KUKA KRL program: wkz1_ab.src, wkz1_ab.dat

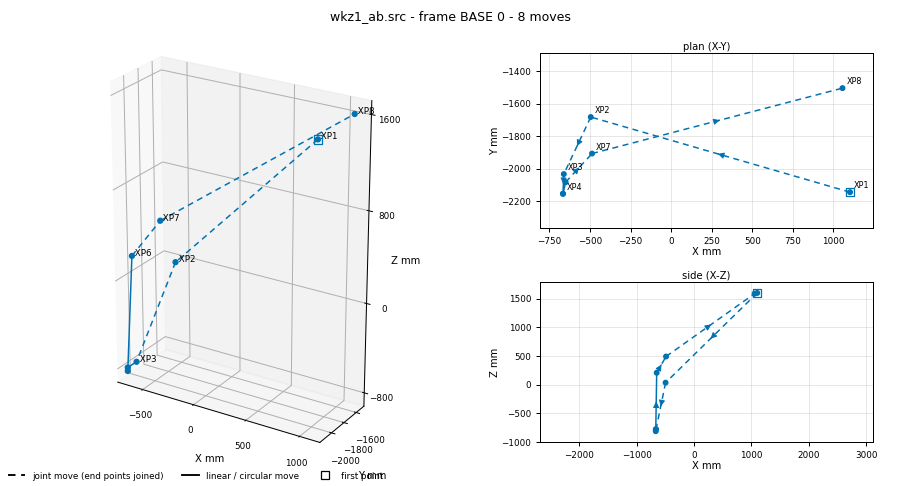
[picture p0: tool path of wkz1_ab.src in frame BASE 0, 8 of 8 moves have a stored position in this frame; points joined in program order, loops and branches not executed]
--- wkz1_ab.src ---
&ACCESS RVO8
&REL 103
&COMMENT DEP_C1
&PARAM DISKPATH = Program/WKZ
DEF WKZ1_AB ( )

;FOLD INI;%{PE}
  ;FOLD BASISTECH INI
    GLOBAL INTERRUPT DECL 3 WHEN $STOPMESS==TRUE DO IR_STOPM ( )
    INTERRUPT ON 3
    BAS (#INITMOV,0 )
  ;ENDFOLD (BASISTECH INI)
;FOLD SPOTTECH INI
USERSPOT(#INIT)
;ENDFOLD (SPOTTECH INI)
;FOLD GRIPPERTECH INI
USER_GRP(0,DUMMY,DUMMY,GDEFAULT)
;ENDFOLD (GRIPPERTECH INI)
  ;FOLD USER INI
    ;Make your modifications here

  ;ENDFOLD (USER INI)
;ENDFOLD (INI)
; Caracterização dos meios de produção:
; Versão Atual:
; 04/05/2013 12:00 Name: P13.090-R6 CHANGES: Deposita C1

chk_w1_wechs_ok ( )              ; CHECK GUN C1

;FOLD PTP P1 Vel=100 % PDAT1 Tool[1]:Gun C1 Base[0];%{PE}%R 8.2.24,%MKUKATPBASIS,%CMOVE,%VPTP,%P 1:PTP, 2:P1, 3:, 5:100, 7:PDAT1
$BWDSTART=FALSE
PDAT_ACT=PPDAT1
FDAT_ACT=FP1
BAS(#PTP_PARAMS,100)
PTP XP1
;ENDFOLD

;FOLD ; START INTERLOCK COM R4;%{PE}%R 8.2.24,%MKUKATPBASIS,%CCOMMENT,%VNORMAL,%P 2:START  INTERLOCK  COM  R4
;ENDFOLD
;FOLD Collision.Monitoring_4_On ;%{PE}%MKUKATPUSER

COLLSTOP( 4, 1 ) ;Interrupt-Controlled

;ENDFOLD

;FOLD WAIT FOR ( NOT IN 161 'DEPOSITO 1 OCUPADO' );%{PE}%R 8.2.24,%MKUKATPBASIS,%CEXT_WAIT_FOR,%VEXT_WAIT_FOR,%P 2:, 4:NOT, 5:$IN, 6:161, 7:DEPOSITO 1 OCUPADO, 9:
WAIT FOR  (  NOT $IN[161] )
;ENDFOLD
;FOLD WAIT FOR ( IN 219 'PLACA DE SUPORTE FUNDIDA' );%{PE}%R 8.2.24,%MKUKATPBASIS,%CEXT_WAIT_FOR,%VEXT_WAIT_FOR,%P 2:, 4:, 5:$IN, 6:219, 7:PLACA DE SUPORTE FUNDIDA, 9:
WAIT FOR  ( $IN[219] )
;ENDFOLD
;FOLD PULSE 167 'Proteção da pinca 1 abrir' State=TRUE Time=0.3 sec;%{PE}%R 8.2.24,%MKUKATPBASIS,%COUT,%VPULSE,%P 2:167, 3:Proteção da pinca 1 abrir, 5:TRUE, 6:, 8:0.3
PULSE($OUT[167], TRUE,0.3)
;ENDFOLD
;FOLD PULSE 184 'Proteção da pinca 3 fechar' State=TRUE Time=0.3 sec;%{PE}%R 8.2.24,%MKUKATPBASIS,%COUT,%VPULSE,%P 2:184, 3:Proteção da pinca 3 fechar, 5:TRUE, 6:, 8:0.3
PULSE($OUT[184], TRUE,0.3)
;ENDFOLD
;FOLD WAIT FOR ( IN 165 'PROTECAO DE PINCA ABERTA' );%{PE}%R 8.2.24,%MKUKATPBASIS,%CEXT_WAIT_FOR,%VEXT_WAIT_FOR,%P 2:, 4:, 5:$IN, 6:165, 7:PROTECAO DE PINCA ABERTA, 9:
WAIT FOR  ( $IN[165] )
;ENDFOLD
;FOLD WAIT FOR ( NOT IN 166 'PROTECAO DE PINCA FECHADA' );%{PE}%R 8.2.24,%MKUKATPBASIS,%CEXT_WAIT_FOR,%VEXT_WAIT_FOR,%P 2:, 4:NOT, 5:$IN, 6:166, 7:PROTECAO DE PINCA FECHADA, 9:
WAIT FOR  (  NOT $IN[166] )
;ENDFOLD
;FOLD WAIT FOR ( IN 182 'PROTECAO DE PINCA FECHADA' );%{PE}%R 8.2.24,%MKUKATPBASIS,%CEXT_WAIT_FOR,%VEXT_WAIT_FOR,%P 2:, 4:, 5:$IN, 6:182, 7:PROTECAO DE PINCA FECHADA, 9:
WAIT FOR  ( $IN[182] )
;ENDFOLD
;FOLD WAIT FOR ( NOT IN 181 'PROTECAO DE PINCA ABERTA' );%{PE}%R 8.2.24,%MKUKATPBASIS,%CEXT_WAIT_FOR,%VEXT_WAIT_FOR,%P 2:, 4:NOT, 5:$IN, 6:181, 7:PROTECAO DE PINCA ABERTA, 9:
WAIT FOR  (  NOT $IN[181] )
;ENDFOLD

;FOLD PTP P2 Vel=100 % PDAT2 Tool[1]:Gun C1 Base[0];%{PE}%R 8.2.24,%MKUKATPBASIS,%CMOVE,%VPTP,%P 1:PTP, 2:P2, 3:, 5:100, 7:PDAT2
$BWDSTART=FALSE
PDAT_ACT=PPDAT2
FDAT_ACT=FP2
BAS(#PTP_PARAMS,100)
PTP XP2
;ENDFOLD
;FOLD PTP P3 Vel=100 % PDAT3 Tool[1]:Gun C1 Base[0];%{PE}%R 8.2.24,%MKUKATPBASIS,%CMOVE,%VPTP,%P 1:PTP, 2:P3, 3:, 5:100, 7:PDAT3
$BWDSTART=FALSE
PDAT_ACT=PPDAT3
FDAT_ACT=FP3
BAS(#PTP_PARAMS,100)
PTP XP3
;ENDFOLD
;FOLD LIN P4 Vel=0.3 m/s CPDAT1 Tool[1]:Gun C1 Base[0];%{PE}%R 8.2.24,%MKUKATPBASIS,%CMOVE,%VLIN,%P 1:LIN, 2:P4, 3:, 5:0.3, 7:CPDAT1
$BWDSTART=FALSE
LDAT_ACT=LCPDAT1
FDAT_ACT=FP4
BAS(#CP_PARAMS,0.3)
LIN XP4
;ENDFOLD

;FOLD ; PONTO DE DEPOSITO PINCA;%{PE}%R 8.2.24,%MKUKATPBASIS,%CCOMMENT,%VNORMAL,%P 2:PONTO  DE  DEPOSITO  PINCA
;ENDFOLD
;FOLD LIN P5 Vel=0.1 m/s CPDAT2 Tool[1]:Gun C1 Base[0];%{PE}%R 8.2.24,%MKUKATPBASIS,%CMOVE,%VLIN,%P 1:LIN, 2:P5, 3:, 5:0.1, 7:CPDAT2
$BWDSTART=FALSE
LDAT_ACT=LCPDAT2
FDAT_ACT=FP5
BAS(#CP_PARAMS,0.1)
LIN XP5
;ENDFOLD

;FOLD WAIT Time=0.5 sec;%{PE}%R 8.2.24,%MKUKATPBASIS,%CWAIT,%VWAIT,%P 3:0.5
WAIT SEC 0.5
;ENDFOLD
;FOLD IBUS OFF;%{PE}%R 8.2.24,%MKUKATPBASIS,%CIBUS,%VMAP,%P 2:#OFF, 3:1
$IBUS_OFF=$IBUS_ON
$IBUS_ON=0
;ENDFOLD
;FOLD WAIT FOR ( IN 161 'DEPOSITO 1 OCUPADO' );%{PE}%R 8.2.24,%MKUKATPBASIS,%CEXT_WAIT_FOR,%VEXT_WAIT_FOR,%P 2:, 4:, 5:$IN, 6:161, 7:DEPOSITO 1 OCUPADO, 9:
WAIT FOR  ( $IN[161] )
;ENDFOLD
;FOLD OUT 223 'DESBLOQUEIA MPS' State=TRUE ;%{PE}%R 8.2.24,%MKUKATPBASIS,%COUT,%VOUTX,%P 2:223, 3:DESBLOQUEIA MPS, 5:TRUE, 6:
$OUT[223]=TRUE
;ENDFOLD
;FOLD OUT 224 'BLOQUEIA MPS' State=FALSE ;%{PE}%R 8.2.24,%MKUKATPBASIS,%COUT,%VOUTX,%P 2:224, 3:BLOQUEIA MPS, 5:FALSE, 6:
$OUT[224]=FALSE
;ENDFOLD
;FOLD WAIT FOR ( IN 217 'MPS DESTRAVADO' );%{PE}%R 8.2.24,%MKUKATPBASIS,%CEXT_WAIT_FOR,%VEXT_WAIT_FOR,%P 2:, 4:, 5:$IN, 6:217, 7:MPS DESTRAVADO, 9:
WAIT FOR  ( $IN[217] )
;ENDFOLD
;FOLD WAIT FOR ( NOT IN 221 'MPS TRAVADO' );%{PE}%R 8.2.24,%MKUKATPBASIS,%CEXT_WAIT_FOR,%VEXT_WAIT_FOR,%P 2:, 4:NOT, 5:$IN, 6:221, 7:MPS TRAVADO, 9:
WAIT FOR  (  NOT $IN[221] )
;ENDFOLD

;FOLD LIN P6 Vel=0.1 m/s CPDAT3 Tool[8]:Tool Changer Base[0];%{PE}%R 8.2.24,%MKUKATPBASIS,%CMOVE,%VLIN,%P 1:LIN, 2:P6, 3:, 5:0.1, 7:CPDAT3
$BWDSTART=FALSE
LDAT_ACT=LCPDAT3
FDAT_ACT=FP6
BAS(#CP_PARAMS,0.1)
LIN XP6
;ENDFOLD

;FOLD WAIT FOR ( NOT IN 219 'PLACA DE SUPORTE FUNDIDA' );%{PE}%R 8.2.24,%MKUKATPBASIS,%CEXT_WAIT_FOR,%VEXT_WAIT_FOR,%P 2:, 4:NOT, 5:$IN, 6:219, 7:PLACA DE SUPORTE FUNDIDA, 9:
WAIT FOR  (  NOT $IN[219] )
;ENDFOLD
;FOLD WAIT FOR ( IN 161 'DEPOSITO 1 OCUPADO' );%{PE}%R 8.2.24,%MKUKATPBASIS,%CEXT_WAIT_FOR,%VEXT_WAIT_FOR,%P 2:, 4:, 5:$IN, 6:161, 7:DEPOSITO 1 OCUPADO, 9:
WAIT FOR  ( $IN[161] )
;ENDFOLD
;FOLD OUT 223 'DESBLOQUEIA MPS' State=FALSE ;%{PE}%R 8.2.24,%MKUKATPBASIS,%COUT,%VOUTX,%P 2:223, 3:DESBLOQUEIA MPS, 5:FALSE, 6:
$OUT[223]=FALSE
;ENDFOLD
;FOLD OUT 224 'BLOQUEIA MPS' State=TRUE ;%{PE}%R 8.2.24,%MKUKATPBASIS,%COUT,%VOUTX,%P 2:224, 3:BLOQUEIA MPS, 5:TRUE, 6:
$OUT[224]=TRUE
;ENDFOLD

;FOLD PTP P7 CONT Vel=100 % PDAT4 Tool[8]:Tool Changer Base[0];%{PE}%R 8.2.24,%MKUKATPBASIS,%CMOVE,%VPTP,%P 1:PTP, 2:P7, 3:C_PTP, 5:100, 7:PDAT4
$BWDSTART=FALSE
PDAT_ACT=PPDAT4
FDAT_ACT=FP7
BAS(#PTP_PARAMS,100)
PTP XP7 C_PTP
;ENDFOLD
;FOLD PTP P8 Vel=100 % PDAT5 Tool[8]:Tool Changer Base[0];%{PE}%R 8.2.24,%MKUKATPBASIS,%CMOVE,%VPTP,%P 1:PTP, 2:P8, 3:, 5:100, 7:PDAT5
$BWDSTART=FALSE
PDAT_ACT=PPDAT5
FDAT_ACT=FP8
BAS(#PTP_PARAMS,100)
PTP XP8
;ENDFOLD

;FOLD ; END INTERLOCK COM R4;%{PE}%R 8.2.24,%MKUKATPBASIS,%CCOMMENT,%VNORMAL,%P 2:END  INTERLOCK  COM  R4
;ENDFOLD
;FOLD Collision.Monitoring_4_Off . ;%{PE}%MKUKATPUSER

COLLSTOP( 4, 2+0 )

;ENDFOLD

;FOLD PULSE 168 'Proteção da pinca 1 fechar' State=TRUE Time=0.3 sec;%{PE}%R 8.2.24,%MKUKATPBASIS,%COUT,%VPULSE,%P 2:168, 3:Proteção da pinca 1 fechar, 5:TRUE, 6:, 8:0.3
PULSE($OUT[168], TRUE,0.3)
;ENDFOLD

;FOLD PULSE 191 'PROTEÇÃO DA PINCA ABRIR' State=TRUE Time=1 sec;%{PE}%R 8.2.24,%MKUKATPBASIS,%COUT,%VPULSE,%P 2:191, 3:PROTEÇÃO DA PINCA ABRIR, 5:TRUE, 6:, 8:1
PULSE($OUT[191], TRUE,1)
;ENDFOLD


END

--- wkz1_ab.dat ---
&ACCESS RVO8
&REL 103
&COMMENT DEP_C1
&PARAM DISKPATH = Program/WKZ
DEFDAT  wkz1_ab
;FOLD EXTERNAL DECLARATIONS;%{PE}%MKUKATPBASIS,%CEXT,%VCOMMON,%P
;FOLD BASISTECH EXT;%{PE}%MKUKATPBASIS,%CEXT,%VEXT,%P
EXT  BAS (BAS_COMMAND  :IN,REAL  :IN )
DECL INT SUCCESS
;ENDFOLD (BASISTECH EXT)
;FOLD USER EXT;%{E}%MKUKATPUSER,%CEXT,%VEXT,%P
;Make your modifications here
;ENDFOLD (USER EXT)
;ENDFOLD (EXTERNAL DECLARATIONS)

;# ============ START PATH : wkz1_ab =============
DECL FDAT Fnew_wkz1_ab_p9={TOOL_NO 1,BASE_NO 0,IPO_FRAME #BASE,POINT2[] " "}
DECL PDAT PP_OLP1={VEL 100.0,ACC 100.0,APO_DIST 0.0}
DECL E6POS Xnew_wkz1_ab_p9={X -683.577026,Y -1624.75195,Z 16.3430004,A 89.2380981,B 24.6753998,C 1.10839999,S 2,T 2}
DECL FDAT Fnew_wkz1_ab_p10={TOOL_NO 1,BASE_NO 0,IPO_FRAME #BASE,POINT2[] " "}
DECL PDAT PP_OLP2={VEL 100.0,ACC 100.0,APO_DIST 0.0}
DECL E6POS Xnew_wkz1_ab_p10={X -661.242004,Y -2032.125,Z -774.536011,A 89.239502,B 24.6767998,C 1.10889995,S 2,T 2}
DECL FDAT Fnew_wkz1_ab_p11={TOOL_NO 1,BASE_NO 0,IPO_FRAME #BASE,POINT2[] " "}
DECL E6POS Xnew_wkz1_ab_p11={X -666.447021,Y -2153.30103,Z -776.817993,A 90.2671967,B 24.6767006,C 1.10870004,S 2,T 2}
DECL LDAT LL_OLP1={VEL 0.300000012,ACC 100.0,APO_DIST 0.0,APO_FAC 0.0,ORI_TYP #VAR,CIRC_TYP #BASE,JERK_FAC 50.0}
DECL FDAT Fnew_wkz1_ab_p12={TOOL_NO 1,BASE_NO 0,IPO_FRAME #BASE,POINT2[] " "}
DECL E6POS Xnew_wkz1_ab_p12={X -666.442993,Y -2153.29907,Z -802.544983,A 90.2675018,B 24.6765003,C 1.10870004,S 2,T 2}
DECL LDAT LL_OLP2={VEL 0.100000001,ACC 100.0,APO_DIST 0.0,APO_FAC 0.0,ORI_TYP #VAR,CIRC_TYP #BASE,JERK_FAC 50.0}
DECL FDAT Fnew_wkz1_ab_p13={TOOL_NO 8,BASE_NO 0,IPO_FRAME #BASE,POINT2[] " "}
DECL E6POS Xnew_wkz1_ab_p13={X -650.067993,Y -2082.00488,Z 209.378998,A -75.2026978,B 0.569100022,C 179.109299,S 2,T 2}
DECL LDAT LL_OLP3={VEL 0.100000001,ACC 100.0,APO_DIST 0.0,APO_FAC 0.0,ORI_TYP #VAR,CIRC_TYP #BASE,JERK_FAC 50.0}
DECL FDAT Fnew_wkz1_ab_p14={TOOL_NO 8,BASE_NO 0,IPO_FRAME #BASE,POINT2[] " "}
DECL PDAT PP_OLP3={VEL 100.0,ACC 100.0,APO_DIST 0.0}
DECL E6POS Xnew_wkz1_ab_p14={X -638.375,Y -2088.72998,Z 595.562988,A -76.4641037,B 0.223000005,C 178.9431,S 2,T 2}
DECL BASIS_SUGG_T LAST_BASIS={POINT1[] "P8                      ",POINT2[] "P8                      ",CP_PARAMS[] "CPDAT3                  ",PTP_PARAMS[] "PDAT5                   ",CONT[] "C_PTP                   ",CP_VEL[] "0.1                     ",PTP_VEL[] "100                     ",SYNC_PARAMS[] "SYNCDAT                 ",SPL_NAME[] "S0                      "}
DECL E6POS XP1={X 1102.26099,Y -2143.50293,Z 1600.37805,A 25.6025009,B 30.4906807,C -50.9274216,S 18,T 10,E1 0.0,E2 0.0,E3 0.0,E4 0.0,E5 0.0,E6 0.0}
DECL FDAT FP1={TOOL_NO 1,BASE_NO 0,IPO_FRAME #BASE,POINT2[] " ",TQ_STATE FALSE}
DECL PDAT PPDAT1={VEL 100.0,ACC 100.0,APO_DIST 100.0,GEAR_JERK 50.0}
DECL E6POS XP2={X -495.25589,Y -1680.54504,Z 37.021389,A 89.43573,B 24.6753292,C 4.75691509,S 18,T 2,E1 0.0,E2 0.0,E3 0.0,E4 0.0,E5 0.0,E6 0.0}
DECL FDAT FP2={TOOL_NO 1,BASE_NO 0,IPO_FRAME #BASE,POINT2[] " ",TQ_STATE FALSE}
DECL PDAT PPDAT2={VEL 100.0,ACC 100.0,APO_DIST 100.0,GEAR_JERK 50.0}
DECL E6POS XP3={X -661.235413,Y -2032.10803,Z -774.536072,A 89.2419434,B 24.6759109,C 1.10841501,S 18,T 2,E1 0.0,E2 0.0,E3 0.0,E4 0.0,E5 0.0,E6 0.0}
DECL FDAT FP3={TOOL_NO 1,BASE_NO 0,IPO_FRAME #BASE,POINT2[] " ",TQ_STATE FALSE}
DECL PDAT PPDAT3={VEL 100.0,ACC 100.0,APO_DIST 100.0,GEAR_JERK 50.0}
DECL E6POS XP4={X -666.448425,Y -2153.28296,Z -776.827881,A 90.2670898,B 24.6758709,C 1.10852802,S 18,T 2,E1 0.0,E2 0.0,E3 0.0,E4 0.0,E5 0.0,E6 0.0}
DECL FDAT FP4={TOOL_NO 1,BASE_NO 0,IPO_FRAME #BASE,POINT2[] " ",TQ_STATE FALSE}
DECL LDAT LCPDAT1={VEL 2.0,ACC 100.0,APO_DIST 100.0,APO_FAC 50.0,AXIS_VEL 100.0,AXIS_ACC 100.0,ORI_TYP #VAR,CIRC_TYP #BASE,JERK_FAC 50.0,GEAR_JERK 50.0,EXAX_IGN 0}
DECL LDAT LCPDAT2={VEL 2.0,ACC 100.0,APO_DIST 100.0,APO_FAC 50.0,AXIS_VEL 100.0,AXIS_ACC 100.0,ORI_TYP #VAR,CIRC_TYP #BASE,JERK_FAC 50.0,GEAR_JERK 50.0,EXAX_IGN 0}
DECL E6POS XP5={X -666.443115,Y -2153.30298,Z -809.122986,A 90.2675629,B 24.6766605,C 1.10863698,S 18,T 2,E1 0.0,E2 0.0,E3 0.0,E4 0.0,E5 0.0,E6 0.0}
DECL FDAT FP5={TOOL_NO 1,BASE_NO 0,IPO_FRAME #BASE,POINT2[] " ",TQ_STATE FALSE}
DECL E6POS XP6={X -650.072083,Y -2082.00806,Z 209.373901,A -75.2018585,B 0.569911122,C 179.109894,S 18,T 2,E1 0.0,E2 0.0,E3 0.0,E4 0.0,E5 0.0,E6 0.0}
DECL FDAT FP6={TOOL_NO 8,BASE_NO 0,IPO_FRAME #BASE,POINT2[] " ",TQ_STATE FALSE}
DECL LDAT LCPDAT3={VEL 2.0,ACC 100.0,APO_DIST 100.0,APO_FAC 50.0,AXIS_VEL 100.0,AXIS_ACC 100.0,ORI_TYP #VAR,CIRC_TYP #BASE,JERK_FAC 50.0,GEAR_JERK 50.0,EXAX_IGN 0}
DECL E6POS XP7={X -487.26239,Y -1905.526,Z 492.567505,A -76.3648682,B 0.161415607,C 173.845001,S 18,T 2,E1 0.0,E2 0.0,E3 0.0,E4 0.0,E5 0.0,E6 0.0}
DECL FDAT FP7={TOOL_NO 8,BASE_NO 0,IPO_FRAME #BASE,POINT2[] " ",TQ_STATE FALSE}
DECL PDAT PPDAT4={VEL 100.0,ACC 100.0,APO_DIST 100.0,APO_MODE #CPTP,GEAR_JERK 50.0}
DECL E6POS XP8={X 1055.87598,Y -1502.40906,Z 1588.43103,A -71.8716202,B -60.8062096,C 178.7379,S 18,T 2,E1 0.0,E2 0.0,E3 0.0,E4 0.0,E5 0.0,E6 0.0}
DECL FDAT FP8={TOOL_NO 8,BASE_NO 0,IPO_FRAME #BASE,POINT2[] " ",TQ_STATE FALSE}
DECL PDAT PPDAT5={VEL 100.0,ACC 100.0,APO_DIST 0.0,APO_MODE #CPTP,GEAR_JERK 50.0}
ENDDAT
